// TIA Portal V19 export
TYPE "LEXCHANGETRAY_typeScanner_monitor"
// stored: Access Published
   STRUCT
      status : "LEXCHANGETRAY_typeScanner_status";
      result : "LEXCHANGETRAY_typeScanner_result";
      simulated { S7_SetPoint := 'True'} : Bool;
   END_STRUCT;
END_TYPE
